{attribute 'qualified_only'}
{attribute 'strict'}
{attribute 'to_string'}
TYPE E_State :
(
	Retract,
	Advance
);
END_TYPE

(* stored: Version 1.1.0.1
   DUT E_State: Id {6b76a1bc-68d4-4416-b877-0ea862f2e1cc} *)
